TYPE UNION_RFID :
UNION
	aArray		: ARRAY[0..63] OF BYTE;
	Number		: UDINT;
END_UNION
END_TYPE

(* stored: Version 1.1.0.1, ProductVersion 3.1.4024.11
   DUT UNION_RFID: Id {df24f2f5-995e-40d9-a3ca-3cd69ddb7cfb} *)
